INTERFACE I_CylinderComponent

END_INTERFACE

(* stored: Version 1.1.0.1, ProductVersion 3.1.4024.12
   Itf I_CylinderComponent: Id {def5f0fb-19d7-4486-9317-9ad0e969cf3f} *)
